TYPE udtYaskawaVFDCmd :
STRUCT
	RunFwd :BOOL;
	RunRev :BOOL;
	ClearFaults :BOOL;	
END_STRUCT
END_TYPE

(* stored: Version 1.1.0.1, ProductVersion 3.1.4020.12
   DUT udtYaskawaVFDCmd: Id {f425c919-2b7b-43e8-8bd4-dfbc96e9589f} *)
